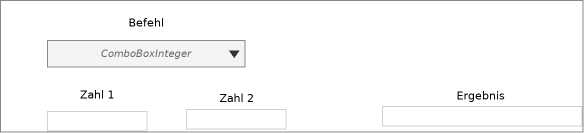
VISUALIZATION Taschenrechner  // 584x133
    ComboBoxInteger (47,40 198x27), variable: MAIN.TaschenRechner.Befehl, text list: 'TaschenrechnerBefehle'
    Textfield (47,111 100x20)
    Label (51,80 93x30), "Zahl 1"
    Textfield (186,109 100x20)
    Label (188,90 98x17), "Zahl 2"
    Textfield (382,106 200x20)
    Label (386,86 189x20), "Ergebnis"
    Label (52,13 189x20), "Befehl"
END_VISUALIZATION

(* stored: Version 1.1.0.1, ProductVersion 3.1.4022.6
   Visu Taschenrechner: Id {529ab607-a3a7-4016-be48-cafee3caa910} *)
